// TIA Portal V18 export
FUNCTION_BLOCK "ER_WN__root_FB"   // FB64, LAD
{ S7_Optimized_Access := 'TRUE' }
VERSION : 0.1
// stored: AutoNumber true, IsIECCheckEnabled false, IsRetainMemResEnabled false, MemoryReserve 100, SetENOAutomatically false, UDAEnableTagReadback false
   VAR_INPUT
      ER_count : Int;
      ACK : Bool;
   END_VAR
   VAR_OUTPUT
      ER_exists : Bool;
   END_VAR
BEGIN

REGION Network 1
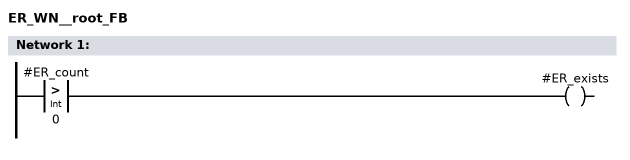
   RUNG wire#powerrail
      { S7_Templates := "SrcType := Int" } GT_Contact(in1 := #ER_count, in2 := 0)
      Coil( #ER_exists )
   END_RUNG
   // the same network as SCL:
   #ER_exists := #ER_count > 0;
END_REGION
END_FUNCTION_BLOCK
